FUNCTION angErrorCalc : LREAL
VAR_INPUT
	 angPosCommand, angPosFdbck:LREAL;
END_VAR
VAR
	angPosDiff:LREAL;
END_VAR

IF(angPosCommand>180) THEN
angPosCommand:=180;
  ELSIF(angPosCommand< -180)THEN
 angPosCommand:=-180;
 END_IF
  angPosDiff:=angPosCommand-angPosFdbck;
  IF(abs(angPosDiff)>180) THEN
    angErrorCalc:= angPosDiff-mySign(angPosDiff)*360;
	RETURN;
  END_IF
  angErrorCalc:= angPosDiff;

END_FUNCTION

(* stored: Version 1.1.0.1, ProductVersion 3.1.4024.12
   POU angErrorCalc: Id {e1f5e2c0-dec8-452b-86d8-234a89a40c54}, SpecialFunc None *)
